TYPE stHMI_MESSENGER :
STRUCT
	currentMsg: POINTER TO MessageDescription;
	activError: POINTER TO MessageDescription;
	bErrorActiv: BOOL;
	bWarnActiv: BOOL;
	MsgCount		: INT := 0;
END_STRUCT
END_TYPE

(* stored: Version 1.1.0.1, ProductVersion 3.1.4026.18
   DUT stHMI_MESSENGER: Id {6935bb95-5d09-4cde-9611-72320afd6960} *)
